TYPE ST_Alarm :
STRUCT
    bAlarmSet: BOOL;
    bAlarmReset: BOOL;
    nStatusLED: E_LedFunction;
    nWarningLED: E_LedFunction;
    nEmergencyLED: E_LedFunction;
    nAcknowledgeLED: E_LedFunction;
    nErrorID: INT;
    sErrorMsg: STRING;
    bAlarmActive: BOOL;
END_STRUCT
END_TYPE

(* stored: Version 1.1.0.1, ProductVersion 3.1.4024.11
   DUT ST_Alarm: Id {7cf4bf56-9560-4e49-afbe-1511a605e206} *)
